(* Logix 5000 project; controller PLC2_Project_5 Emulate 5570 rev 20.11; software revision 20.00 *)

TASK MainTask (continuous, watchdog 500 ms) : MainProgram

MODULES
   Local : Emulate 5570 (ICP 1, rev 20.11)
END_MODULES

PROGRAM MainProgram   (* main routine MainRoutine *)
VAR
   in_rotameterBit : BOOL; {access Read Only}
   Oil_Flowrate : REAL; {access Read Only}
   Oil_TempTimerValue : DINT; {access Read Only}
   Oil_TimeSinceLastPuls : REAL; {access Read Only}
   RotameterBit : BOOL; {access Read Only}
   sim_rotameter : TIMER := (PRE := 1000);
   Timer_Rotameter : TIMER := (PRE := 99999); {access Read Only}
END_VAR

ROUTINE Control   (* ladder *)
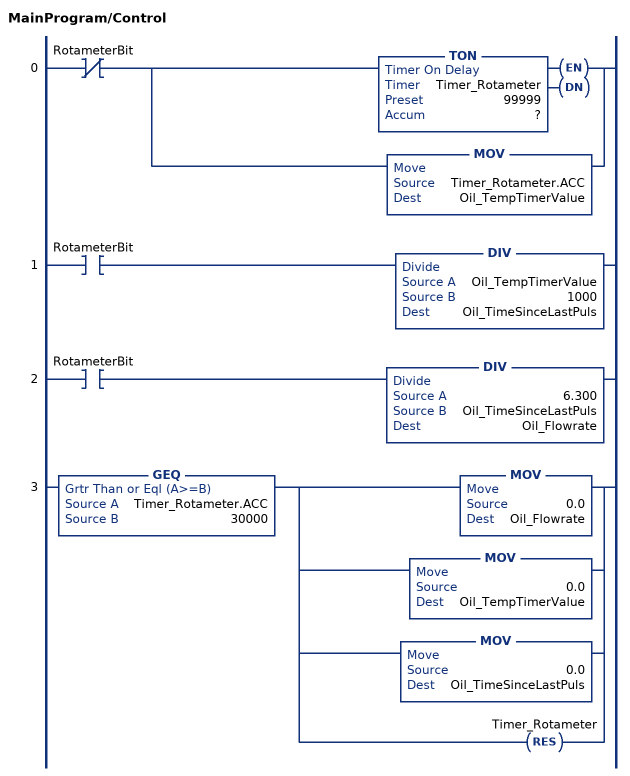
   0: XIO(RotameterBit)[TON(Timer_Rotameter,?,?) ,MOV(Timer_Rotameter.ACC,Oil_TempTimerValue) ];
   1: XIC(RotameterBit)DIV(Oil_TempTimerValue,1000,Oil_TimeSinceLastPuls);
   2: XIC(RotameterBit)DIV(6.300,Oil_TimeSinceLastPuls,Oil_Flowrate);
   3: GEQ(Timer_Rotameter.ACC,30000)[MOV(0.0,Oil_Flowrate) ,MOV(0.0,Oil_TempTimerValue) ,MOV(0.0,Oil_TimeSinceLastPuls) ,RES(Timer_Rotameter) ];
END_ROUTINE

ROUTINE Input_Output   (* ladder *)
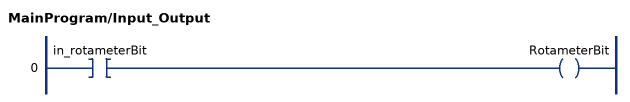
   0: XIC(in_rotameterBit)OTE(RotameterBit);
END_ROUTINE

ROUTINE MainRoutine   (* ladder *)
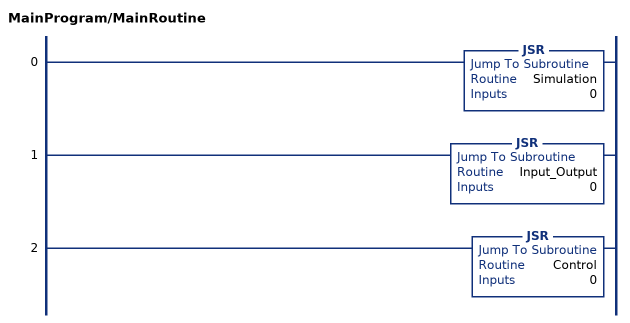
   0: JSR(Simulation,0);
   1: JSR(Input_Output,0);
   2: JSR(Control,0);
END_ROUTINE

ROUTINE Simulation   (* ladder *)
// Simulates a rotameter input.
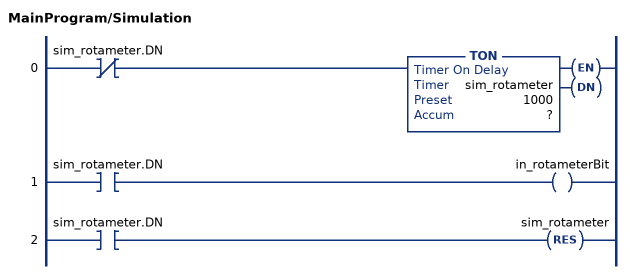
   0: XIO(sim_rotameter.DN)TON(sim_rotameter,?,?);
   1: XIC(sim_rotameter.DN)OTE(in_rotameterBit);
   2: XIC(sim_rotameter.DN)RES(sim_rotameter);
END_ROUTINE
END_PROGRAM
